PROGRAM Lids
VAR
	
	IsLidAtPlaceTrig: F_TRIG;
END_VAR

CASE gvl.CurrentLidsState OF
	LidStates.WaitingToStart:
	gvl.LidClamperRiserMotor:=FALSE;
	gvl.LidClampMotor:=FALSE;
	GVL.LidConveyorMotor:=FALSE;
	LidStates.LocatingInPlace:
	gvl.LidConveyorMotor:=TRUE;
	IsLidAtPlaceTrig(CLK:=gvl.IsLidAtPlace , Q=> );
	
	IF 	IsLidAtPlaceTrig.Q THEN
		gvl.LidConveyorMotor:=FALSE;
		gvl.LidClampMotor:=TRUE;
		gvl.CurrentLidsState:=LidStates.PickingAndPlacing;
	END_IF
	LidStates.PickingAndPlacing:
	
	IF gvl.IsBaseAtPlace THEN
		gvl.CurrentLidsState:=LidStates.LocatingInPlace;
	END_IF
	
	LidStates.Stop:
	
	gvl.LidClamperRiserMotor:=FALSE;
	gvl.LidClampMotor:=FALSE;
	GVL.LidConveyorMotor:=FALSE;
	
	
END_CASE

END_PROGRAM

(* stored: Version 1.1.0.1, ProductVersion 3.1.4024.9
   POU Lids: Id {13374413-e6f4-437b-92d8-ee07c26b3b51}, SpecialFunc None *)
